// TIA Portal V18 export
DATA_BLOCK "AHUOpModes"   // DB102
{ S7_Optimized_Access := 'FALSE' }
VERSION : 0.1
// stored: AutoNumber false, DBAccessibleFromOPCUA true, IsOnlyStoredInLoadMemory false, IsWriteProtectedInAS false
   VAR RETAIN
      OpModes { S7_SetPoint := 'True'} : "UDT_AHUsMode";
   END_VAR
BEGIN
   OpModes.cPreselectedOpModePLC[1..3] := 0;
   OpModes.cSchedulerTargetUnitOpMode[1..2] := 3;
   OpModes.cSchedulerTargetUnitOpMode[3] := 0;
END_DATA_BLOCK
